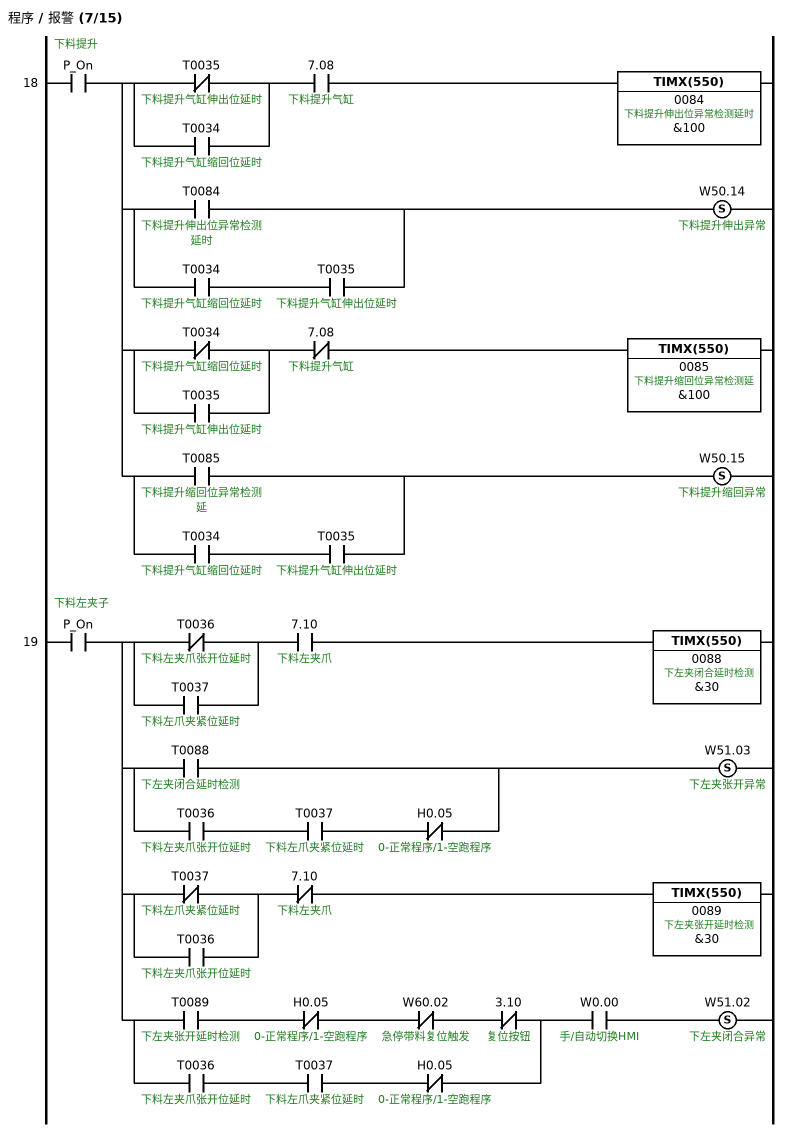
; rung 18: 下料提升
LD P_On
OUT TR0
LDNOT T0035  ; 下料提升气缸伸出位延时
OR T0034  ; 下料提升气缸缩回位延时
ANDLD
AND 7.08  ; 下料提升气缸
TIMX(550) 0084 &100  ; 下料提升伸出位异常检测延时
LD TR0
LD T0084  ; 下料提升伸出位异常检测延时
LD T0034  ; 下料提升气缸缩回位延时
AND T0035  ; 下料提升气缸伸出位延时
ORLD
ANDLD
SET W50.14  ; 下料提升伸出异常
LD TR0
LDNOT T0034  ; 下料提升气缸缩回位延时
OR T0035  ; 下料提升气缸伸出位延时
ANDLD
ANDNOT 7.08  ; 下料提升气缸
TIMX(550) 0085 &100  ; 下料提升缩回位异常检测延
LD TR0
LD T0085  ; 下料提升缩回位异常检测延
LD T0034  ; 下料提升气缸缩回位延时
AND T0035  ; 下料提升气缸伸出位延时
ORLD
ANDLD
SET W50.15  ; 下料提升缩回异常
; rung 19: 下料左夹子
LD P_On
OUT TR0
LDNOT T0036  ; 下料左夹爪张开位延时
OR T0037  ; 下料左爪夹紧位延时
ANDLD
AND 7.10  ; 下料左夹爪
TIMX(550) 0088 &30  ; 下左夹闭合延时检测
LD TR0
LD T0088  ; 下左夹闭合延时检测
LD T0036  ; 下料左夹爪张开位延时
AND T0037  ; 下料左爪夹紧位延时
ANDNOT H0.05  ; 0-正常程序/1-空跑程序
ORLD
ANDLD
SET W51.03  ; 下左夹张开异常
LD TR0
LDNOT T0037  ; 下料左爪夹紧位延时
OR T0036  ; 下料左夹爪张开位延时
ANDLD
ANDNOT 7.10  ; 下料左夹爪
TIMX(550) 0089 &30  ; 下左夹张开延时检测
LD TR0
LD T0089  ; 下左夹张开延时检测
ANDNOT H0.05  ; 0-正常程序/1-空跑程序
ANDNOT W60.02  ; 急停带料复位触发
ANDNOT 3.10  ; 复位按钮
LD T0036  ; 下料左夹爪张开位延时
AND T0037  ; 下料左爪夹紧位延时
ANDNOT H0.05  ; 0-正常程序/1-空跑程序
ORLD
ANDLD
AND W0.00  ; 手/自动切换HMI
SET W51.02  ; 下左夹闭合异常

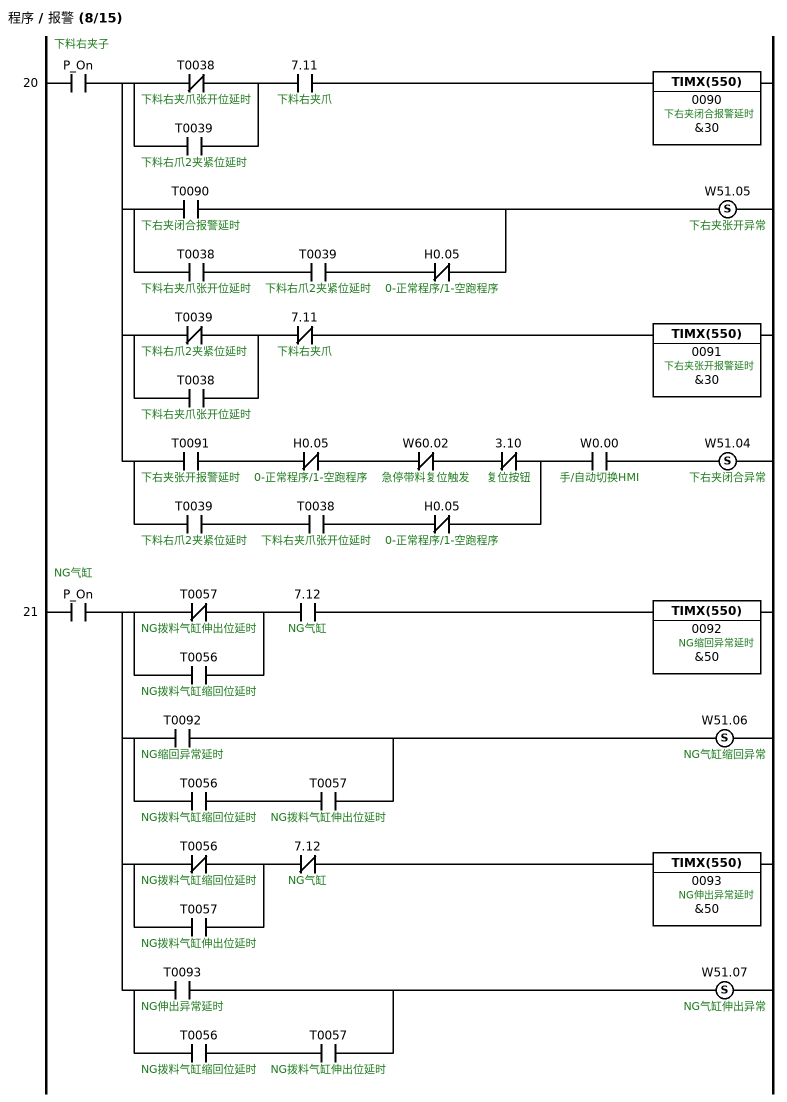
; rung 20: 下料右夹子
LD P_On
OUT TR0
LDNOT T0038  ; 下料右夹爪张开位延时
OR T0039  ; 下料右爪2夹紧位延时
ANDLD
AND 7.11  ; 下料右夹爪
TIMX(550) 0090 &30  ; 下右夹闭合报警延时
LD TR0
LD T0090  ; 下右夹闭合报警延时
LD T0038  ; 下料右夹爪张开位延时
AND T0039  ; 下料右爪2夹紧位延时
ANDNOT H0.05  ; 0-正常程序/1-空跑程序
ORLD
ANDLD
SET W51.05  ; 下右夹张开异常
LD TR0
LDNOT T0039  ; 下料右爪2夹紧位延时
OR T0038  ; 下料右夹爪张开位延时
ANDLD
ANDNOT 7.11  ; 下料右夹爪
TIMX(550) 0091 &30  ; 下右夹张开报警延时
LD TR0
LD T0091  ; 下右夹张开报警延时
ANDNOT H0.05  ; 0-正常程序/1-空跑程序
ANDNOT W60.02  ; 急停带料复位触发
ANDNOT 3.10  ; 复位按钮
LD T0039  ; 下料右爪2夹紧位延时
AND T0038  ; 下料右夹爪张开位延时
ANDNOT H0.05  ; 0-正常程序/1-空跑程序
ORLD
ANDLD
AND W0.00  ; 手/自动切换HMI
SET W51.04  ; 下右夹闭合异常
; rung 21: NG气缸
LD P_On
OUT TR0
LDNOT T0057  ; NG拨料气缸伸出位延时
OR T0056  ; NG拨料气缸缩回位延时
ANDLD
AND 7.12  ; NG气缸
TIMX(550) 0092 &50  ; NG缩回异常延时
LD TR0
LD T0092  ; NG缩回异常延时
LD T0056  ; NG拨料气缸缩回位延时
AND T0057  ; NG拨料气缸伸出位延时
ORLD
ANDLD
SET W51.06  ; NG气缸缩回异常
LD TR0
LDNOT T0056  ; NG拨料气缸缩回位延时
OR T0057  ; NG拨料气缸伸出位延时
ANDLD
ANDNOT 7.12  ; NG气缸
TIMX(550) 0093 &50  ; NG伸出异常延时
LD TR0
LD T0093  ; NG伸出异常延时
LD T0056  ; NG拨料气缸缩回位延时
AND T0057  ; NG拨料气缸伸出位延时
ORLD
ANDLD
SET W51.07  ; NG气缸伸出异常

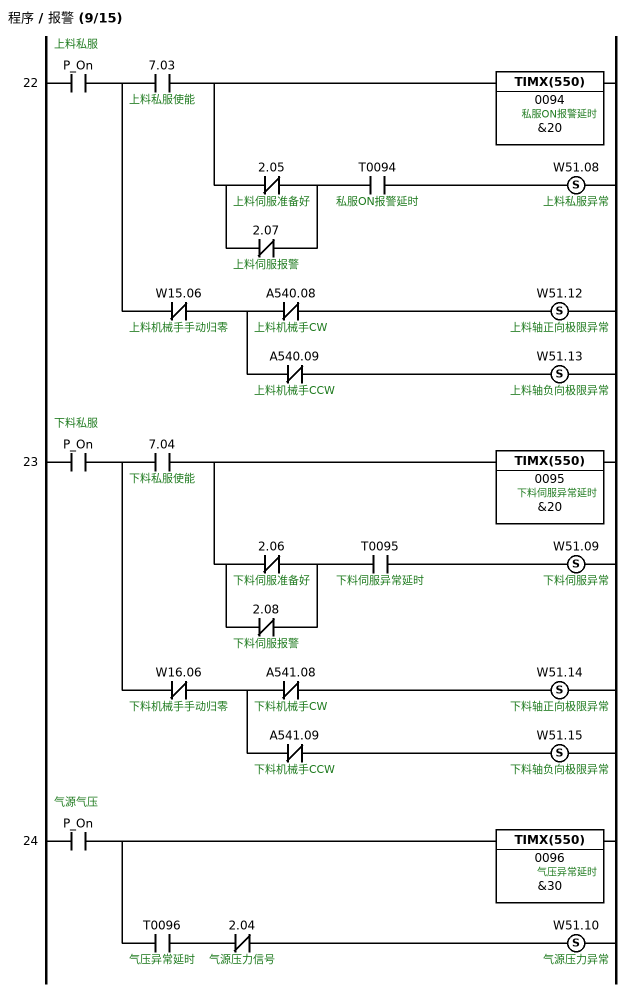
; rung 22: 上料私服
LD P_On
OUT TR0
AND 7.03  ; 上料私服使能
TIMX(550) 0094 &20  ; 私服ON报警延时
LDNOT 2.05  ; 上料伺服准备好
ORNOT 2.07  ; 上料伺服报警
ANDLD
AND T0094  ; 私服ON报警延时
SET W51.08  ; 上料私服异常
LD TR0
ANDNOT W15.06  ; 上料机械手手动归零
OUT TR0
ANDNOT A540.08  ; 上料机械手CW
SET W51.12  ; 上料轴正向极限异常
LD TR0
ANDNOT A540.09  ; 上料机械手CCW
SET W51.13  ; 上料轴负向极限异常
; rung 23: 下料私服
LD P_On
OUT TR0
AND 7.04  ; 下料私服使能
TIMX(550) 0095 &20  ; 下料伺服异常延时
LDNOT 2.06  ; 下料伺服准备好
ORNOT 2.08  ; 下料伺服报警
ANDLD
AND T0095  ; 下料伺服异常延时
SET W51.09  ; 下料伺服异常
LD TR0
ANDNOT W16.06  ; 下料机械手手动归零
OUT TR0
ANDNOT A541.08  ; 下料机械手CW
SET W51.14  ; 下料轴正向极限异常
LD TR0
ANDNOT A541.09  ; 下料机械手CCW
SET W51.15  ; 下料轴负向极限异常
; rung 24: 气源气压
LD P_On
TIMX(550) 0096 &30  ; 气压异常延时
AND T0096  ; 气压异常延时
ANDNOT 2.04  ; 气源压力信号
SET W51.10  ; 气源压力异常

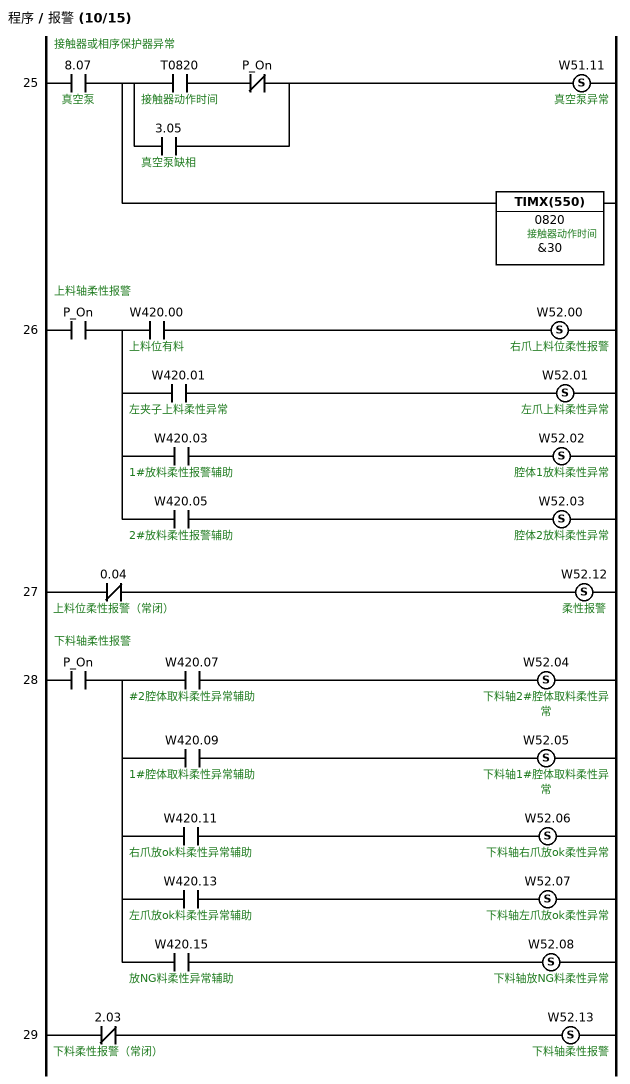
; rung 25: 接触器或相序保护器异常
LD 8.07  ; 真空泵
OUT TR0
LD T0820  ; 接触器动作时间
ANDNOT P_On
OR 3.05  ; 真空泵缺相
ANDLD
SET W51.11  ; 真空泵异常
LD TR0
TIMX(550) 0820 &30  ; 接触器动作时间
; rung 26: 上料轴柔性报警
LD P_On
OUT TR0
AND W420.00  ; 上料位有料
SET W52.00  ; 右爪上料位柔性报警
LD TR0
AND W420.01  ; 左夹子上料柔性异常
SET W52.01  ; 左爪上料柔性异常
LD TR0
AND W420.03  ; 1#放料柔性报警辅助
SET W52.02  ; 腔体1放料柔性异常
LD TR0
AND W420.05  ; 2#放料柔性报警辅助
SET W52.03  ; 腔体2放料柔性异常
; rung 27
LDNOT 0.04  ; 上料位柔性报警（常闭）
SET W52.12  ; 柔性报警
; rung 28: 下料轴柔性报警
LD P_On
OUT TR0
AND W420.07  ; #2腔体取料柔性异常辅助
SET W52.04  ; 下料轴2#腔体取料柔性异常
LD TR0
AND W420.09  ; 1#腔体取料柔性异常辅助
SET W52.05  ; 下料轴1#腔体取料柔性异常
LD TR0
AND W420.11  ; 右爪放ok料柔性异常辅助
SET W52.06  ; 下料轴右爪放ok柔性异常
LD TR0
AND W420.13  ; 左爪放ok料柔性异常辅助
SET W52.07  ; 下料轴左爪放ok柔性异常
LD TR0
AND W420.15  ; 放NG料柔性异常辅助
SET W52.08  ; 下料轴放NG料柔性异常
; rung 29
LDNOT 2.03  ; 下料柔性报警（常闭）
SET W52.13  ; 下料轴柔性报警

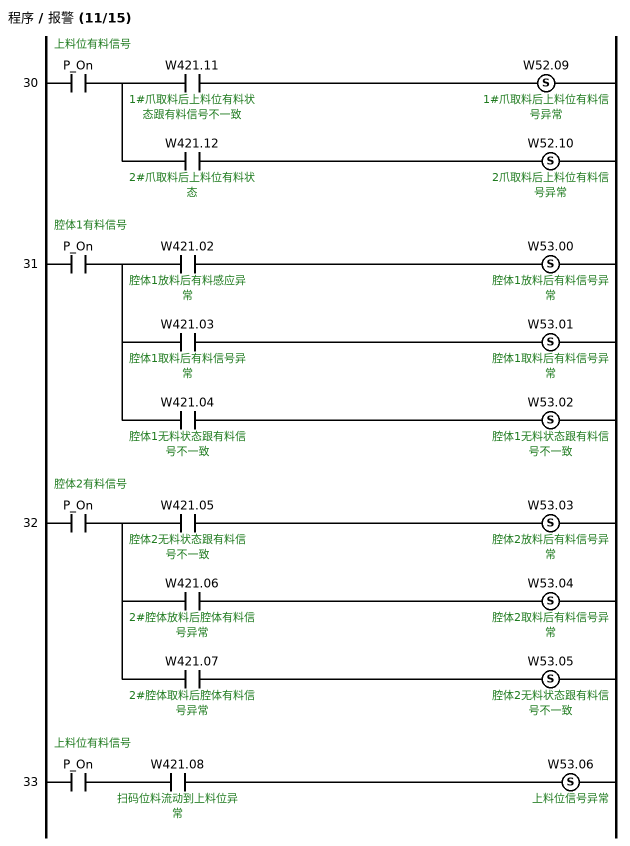
; rung 30: 上料位有料信号
LD P_On
OUT TR0
AND W421.11  ; 1#爪取料后上料位有料状态跟有料信号不一致
SET W52.09  ; 1#爪取料后上料位有料信号异常
LD TR0
AND W421.12  ; 2#爪取料后上料位有料状态
SET W52.10  ; 2爪取料后上料位有料信号异常
; rung 31: 腔体1有料信号
LD P_On
OUT TR0
AND W421.02  ; 腔体1放料后有料感应异常
SET W53.00  ; 腔体1放料后有料信号异常
LD TR0
AND W421.03  ; 腔体1取料后有料信号异常
SET W53.01  ; 腔体1取料后有料信号异常
LD TR0
AND W421.04  ; 腔体1无料状态跟有料信号不一致
SET W53.02  ; 腔体1无料状态跟有料信号不一致
; rung 32: 腔体2有料信号
LD P_On
OUT TR0
AND W421.05  ; 腔体2无料状态跟有料信号不一致
SET W53.03  ; 腔体2放料后有料信号异常
LD TR0
AND W421.06  ; 2#腔体放料后腔体有料信号异常
SET W53.04  ; 腔体2取料后有料信号异常
LD TR0
AND W421.07  ; 2#腔体取料后腔体有料信号异常
SET W53.05  ; 腔体2无料状态跟有料信号不一致
; rung 33: 上料位有料信号
LD P_On
AND W421.08  ; 扫码位料流动到上料位异常
SET W53.06  ; 上料位信号异常

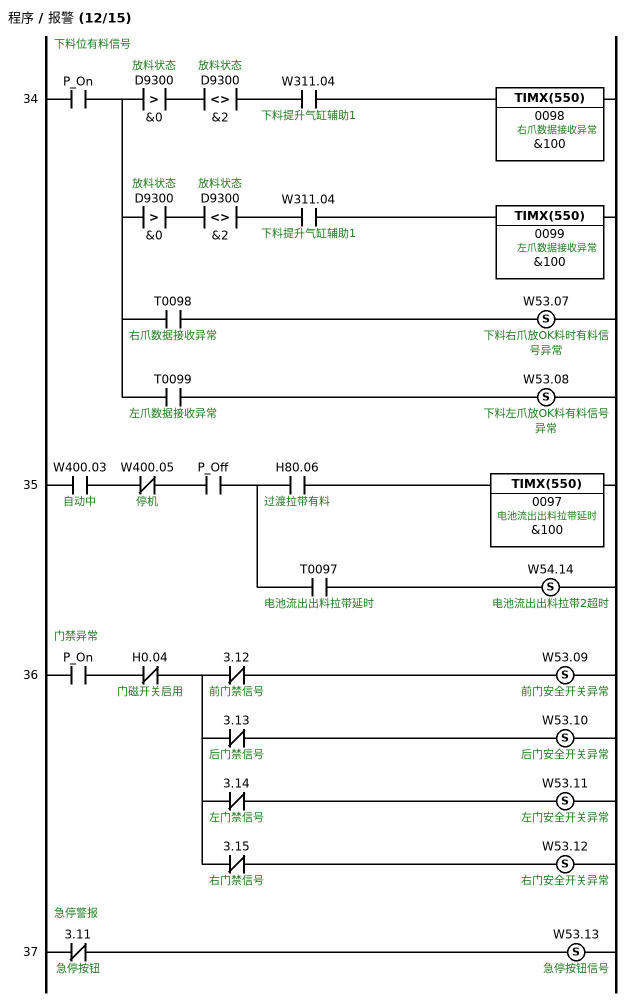
; rung 34: 下料位有料信号
LD P_On
OUT TR0
AND>(320) D9300 &0  ; 放料状态
AND<>(305) D9300 &2  ; 放料状态
AND W311.04  ; 下料提升气缸辅助1
TIMX(550) 0098 &100  ; 右爪数据接收异常
LD TR0
AND>(320) D9300 &0  ; 放料状态
AND<>(305) D9300 &2  ; 放料状态
AND W311.04  ; 下料提升气缸辅助1
TIMX(550) 0099 &100  ; 左爪数据接收异常
LD TR0
AND T0098  ; 右爪数据接收异常
SET W53.07  ; 下料右爪放OK料时有料信号异常
LD TR0
AND T0099  ; 左爪数据接收异常
SET W53.08  ; 下料左爪放OK料有料信号异常
; rung 35
LD W400.03  ; 自动中
ANDNOT W400.05  ; 停机
AND P_Off
OUT TR0
AND H80.06  ; 过渡拉带有料
TIMX(550) 0097 &100  ; 电池流出出料拉带延时
LD TR0
AND T0097  ; 电池流出出料拉带延时
SET W54.14  ; 电池流出出料拉带2超时
; rung 36: 门禁异常
LD P_On
ANDNOT H0.04  ; 门磁开关启用
OUT TR0
ANDNOT 3.12  ; 前门禁信号
SET W53.09  ; 前门安全开关异常
LD TR0
ANDNOT 3.13  ; 后门禁信号
SET W53.10  ; 后门安全开关异常
LD TR0
ANDNOT 3.14  ; 左门禁信号
SET W53.11  ; 左门安全开关异常
LD TR0
ANDNOT 3.15  ; 右门禁信号
SET W53.12  ; 右门安全开关异常
; rung 37: 急停警报
LDNOT 3.11  ; 急停按钮
SET W53.13  ; 急停按钮信号

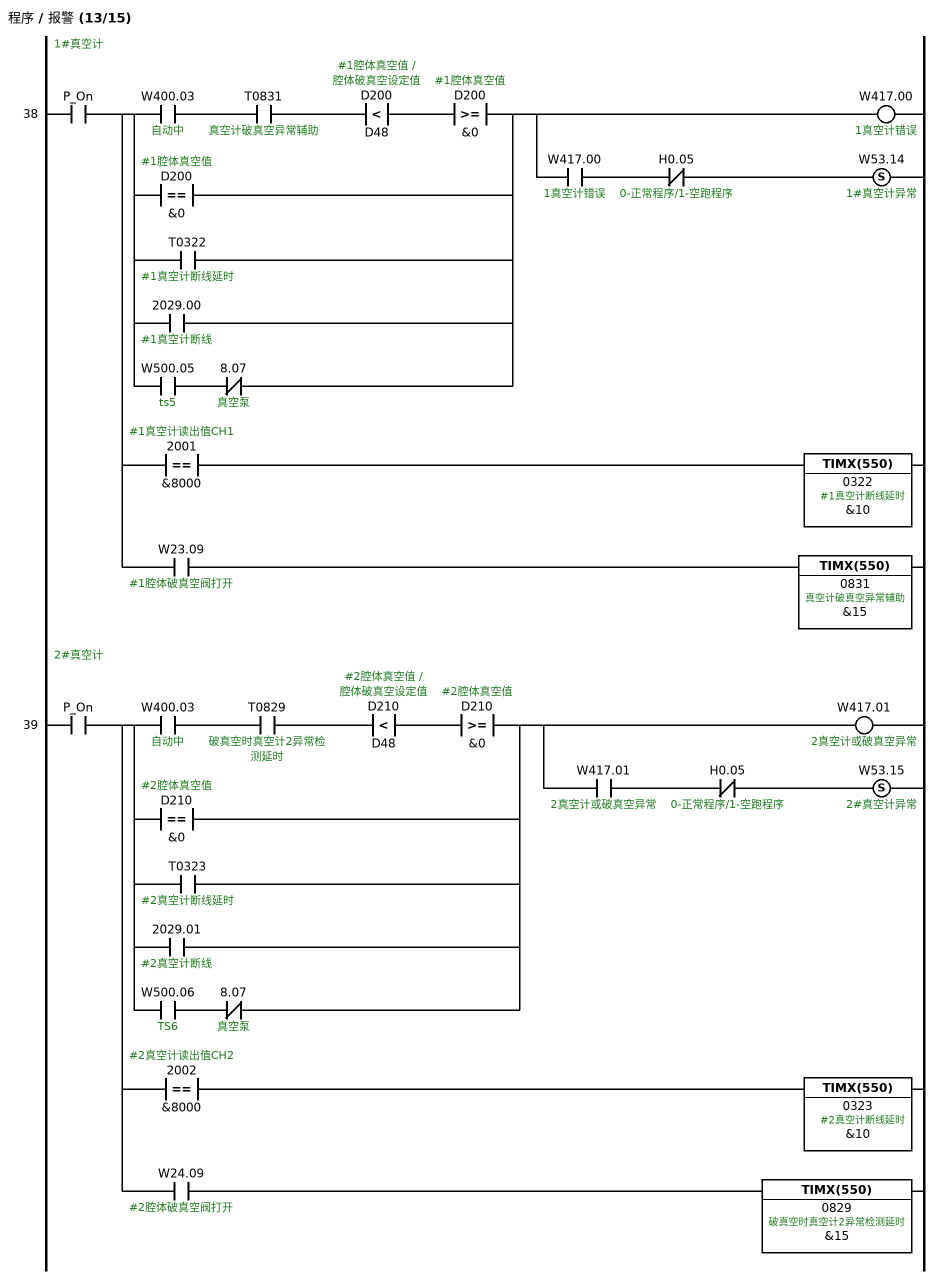
; rung 38: 1#真空计
LD P_On
OUT TR0
LD W400.03  ; 自动中
AND T0831  ; 真空计破真空异常辅助
AND<F(331) D200 D48  ; #1腔体真空值, 腔体破真空设定值
AND>=F(334) D200 &0  ; #1腔体真空值
OR=F(329) D200 &0  ; #1腔体真空值
OR T0322  ; #1真空计断线延时
OR 2029.00  ; #1真空计断线
LD W500.05  ; ts5
ANDNOT 8.07  ; 真空泵
ORLD
ANDLD
OUT W417.00  ; 1真空计错误
AND W417.00  ; 1真空计错误
ANDNOT H0.05  ; 0-正常程序/1-空跑程序
SET W53.14  ; 1#真空计异常
LD TR0
AND=(300) 2001 &8000  ; #1真空计读出值CH1
TIMX(550) 0322 &10  ; #1真空计断线延时
LD TR0
AND W23.09  ; #1腔体破真空阀打开
TIMX(550) 0831 &15  ; 真空计破真空异常辅助
; rung 39: 2#真空计
LD P_On
OUT TR0
LD W400.03  ; 自动中
AND T0829  ; 破真空时真空计2异常检测延时
AND<F(331) D210 D48  ; #2腔体真空值, 腔体破真空设定值
AND>=F(334) D210 &0  ; #2腔体真空值
OR=F(329) D210 &0  ; #2腔体真空值
OR T0323  ; #2真空计断线延时
OR 2029.01  ; #2真空计断线
LD W500.06  ; TS6
ANDNOT 8.07  ; 真空泵
ORLD
ANDLD
OUT W417.01  ; 2真空计或破真空异常
AND W417.01  ; 2真空计或破真空异常
ANDNOT H0.05  ; 0-正常程序/1-空跑程序
SET W53.15  ; 2#真空计异常
LD TR0
AND=(300) 2002 &8000  ; #2真空计读出值CH2
TIMX(550) 0323 &10  ; #2真空计断线延时
LD TR0
AND W24.09  ; #2腔体破真空阀打开
TIMX(550) 0829 &15  ; 破真空时真空计2异常检测延时

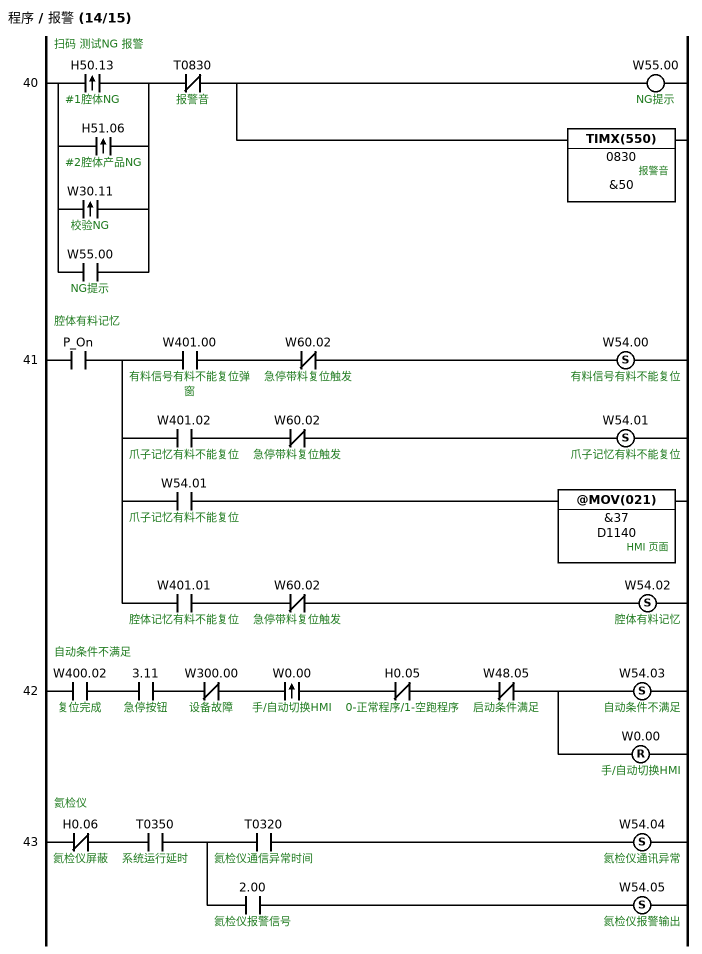
; rung 40: 扫码 测试NG 报警
@LD H50.13  ; #1腔体NG
@OR H51.06  ; #2腔体产品NG
@OR W30.11  ; 校验NG
OR W55.00  ; NG提示
ANDNOT T0830  ; 报警音
OUT W55.00  ; NG提示
TIMX(550) 0830 &50  ; 报警音
; rung 41: 腔体有料记忆
LD P_On
OUT TR0
AND W401.00  ; 有料信号有料不能复位弹窗
ANDNOT W60.02  ; 急停带料复位触发
SET W54.00  ; 有料信号有料不能复位
LD TR0
AND W401.02  ; 爪子记忆有料不能复位
ANDNOT W60.02  ; 急停带料复位触发
SET W54.01  ; 爪子记忆有料不能复位
LD TR0
AND W54.01  ; 爪子记忆有料不能复位
@MOV(021) &37 D1140  ; HMI 页面
LD TR0
AND W401.01  ; 腔体记忆有料不能复位
ANDNOT W60.02  ; 急停带料复位触发
SET W54.02  ; 腔体有料记忆
; rung 42: 自动条件不满足
LD W400.02  ; 复位完成
AND 3.11  ; 急停按钮
ANDNOT W300.00  ; 设备故障
@AND W0.00  ; 手/自动切换HMI
ANDNOT H0.05  ; 0-正常程序/1-空跑程序
ANDNOT W48.05  ; 启动条件满足
SET W54.03  ; 自动条件不满足
RSET W0.00  ; 手/自动切换HMI
; rung 43: 氦检仪
LDNOT H0.06  ; 氦检仪屏蔽
AND T0350  ; 系统运行延时  // 2018/7/25 由常通改为T350，避免开机氦检仪报警
OUT TR0
AND T0320  ; 氦检仪通信异常时间
SET W54.04  ; 氦检仪通讯异常
LD TR0
AND 2.00  ; 氦检仪报警信号
SET W54.05  ; 氦检仪报警输出

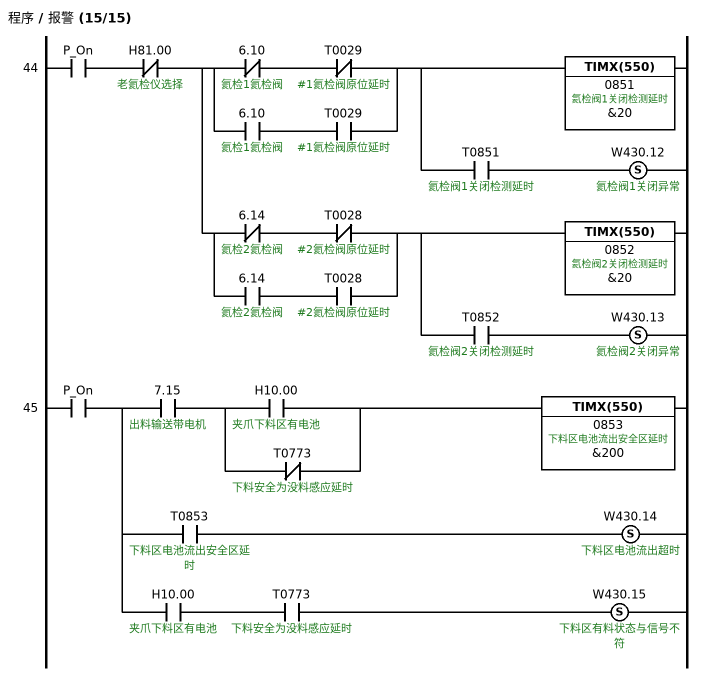
; rung 44
LD P_On
ANDNOT H81.00  ; 老氦检仪选择
OUT TR0
LDNOT 6.10  ; 氦检1氦检阀
ANDNOT T0029  ; #1氦检阀原位延时
LD 6.10  ; 氦检1氦检阀
AND T0029  ; #1氦检阀原位延时
ORLD
ANDLD
TIMX(550) 0851 &20  ; 氦检阀1关闭检测延时
AND T0851  ; 氦检阀1关闭检测延时
SET W430.12  ; 氦检阀1关闭异常
LD TR0
LDNOT 6.14  ; 氦检2氦检阀
ANDNOT T0028  ; #2氦检阀原位延时
LD 6.14  ; 氦检2氦检阀
AND T0028  ; #2氦检阀原位延时
ORLD
ANDLD
TIMX(550) 0852 &20  ; 氦检阀2关闭检测延时
AND T0852  ; 氦检阀2关闭检测延时
SET W430.13  ; 氦检阀2关闭异常
; rung 45
LD P_On
OUT TR0
AND 7.15  ; 出料输送带电机
LD H10.00  ; 夹爪下料区有电池
ORNOT T0773  ; 下料安全为没料感应延时
ANDLD
TIMX(550) 0853 &200  ; 下料区电池流出安全区延时
LD TR0
AND T0853  ; 下料区电池流出安全区延时
SET W430.14  ; 下料区电池流出超时
LD TR0
AND H10.00  ; 夹爪下料区有电池
AND T0773  ; 下料安全为没料感应延时
SET W430.15  ; 下料区有料状态与信号不符

### Section 传感器屏蔽及延时

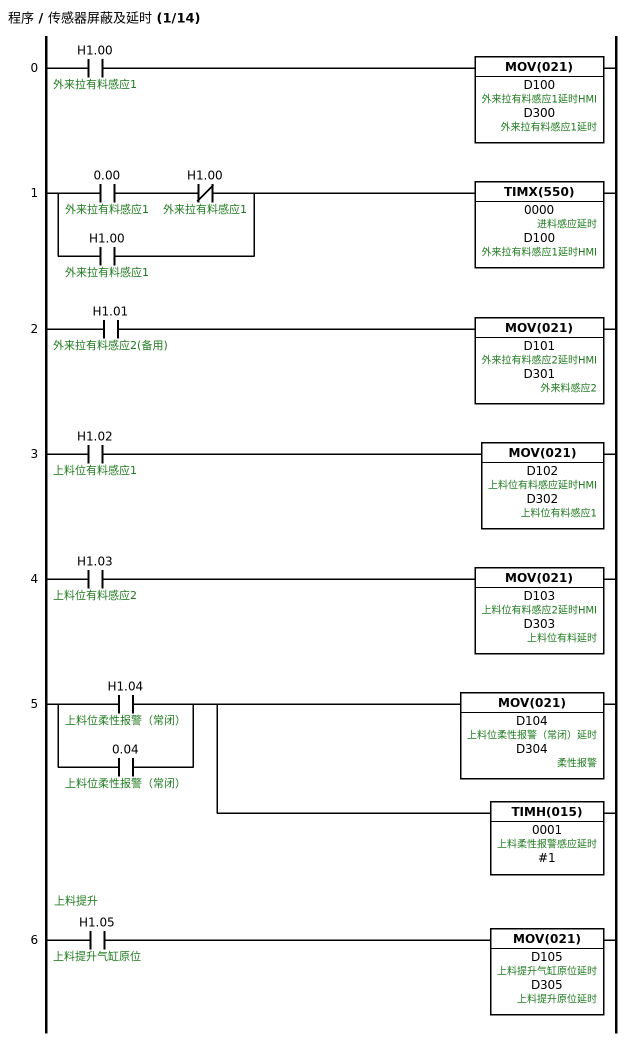
; rung 0
LD H1.00  ; 外来拉有料感应1
MOV(021) D100 D300  ; 外来拉有料感应1延时HMI, 外来拉有料感应1延时
; rung 1
LD 0.00  ; 外来拉有料感应1
ANDNOT H1.00  ; 外来拉有料感应1
OR H1.00  ; 外来拉有料感应1
TIMX(550) 0000 D100  ; 外来拉有料感应1延时HMI, 进料感应延时
; rung 2
LD H1.01  ; 外来拉有料感应2(备用)
MOV(021) D101 D301  ; 外来拉有料感应2延时HMI, 外来料感应2
; rung 3
LD H1.02  ; 上料位有料感应1
MOV(021) D102 D302  ; 上料位有料感应延时HMI, 上料位有料感应1
; rung 4
LD H1.03  ; 上料位有料感应2
MOV(021) D103 D303  ; 上料位有料感应2延时HMI, 上料位有料延时
; rung 5
LD H1.04  ; 上料位柔性报警（常闭）
OR 0.04  ; 上料位柔性报警（常闭）
MOV(021) D104 D304  ; 上料位柔性报警（常闭）延时, 柔性报警
TIMH(015) 0001 #1  ; 上料柔性报警感应延时
; rung 6: 上料提升
LD H1.05  ; 上料提升气缸原位
MOV(021) D105 D305  ; 上料提升气缸原位延时, 上料提升原位延时

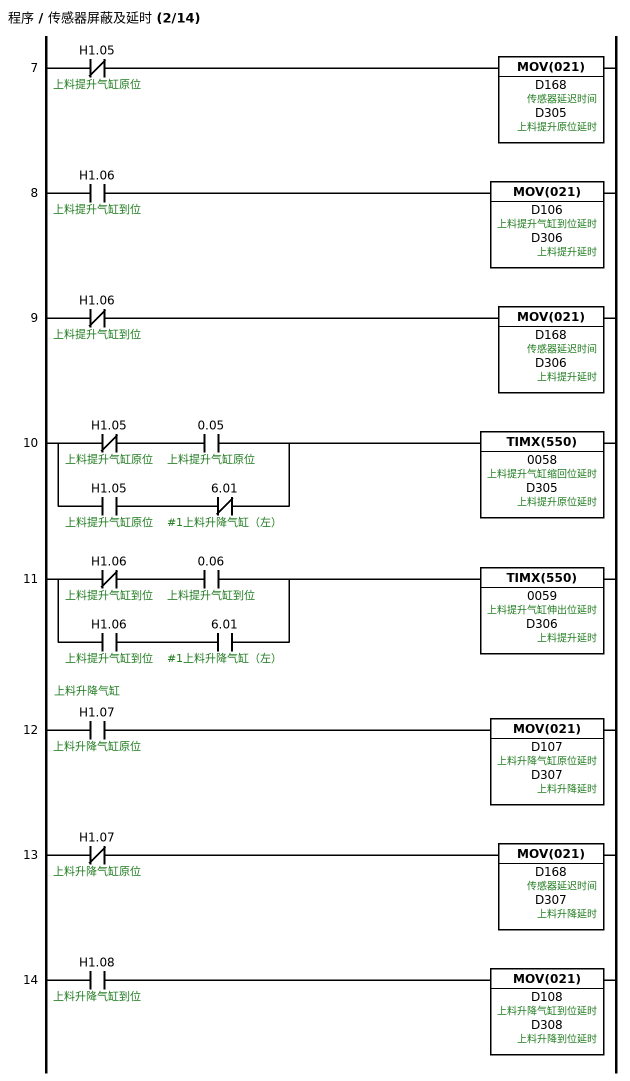
; rung 7
LDNOT H1.05  ; 上料提升气缸原位
MOV(021) D168 D305  ; 传感器延迟时间, 上料提升原位延时
; rung 8
LD H1.06  ; 上料提升气缸到位
MOV(021) D106 D306  ; 上料提升气缸到位延时, 上料提升延时
; rung 9
LDNOT H1.06  ; 上料提升气缸到位
MOV(021) D168 D306  ; 传感器延迟时间, 上料提升延时
; rung 10
LDNOT H1.05  ; 上料提升气缸原位
AND 0.05  ; 上料提升气缸原位
LD H1.05  ; 上料提升气缸原位
ANDNOT 6.01  ; #1上料升降气缸（左）
ORLD
TIMX(550) 0058 D305  ; 上料提升原位延时, 上料提升气缸缩回位延时
; rung 11
LDNOT H1.06  ; 上料提升气缸到位
AND 0.06  ; 上料提升气缸到位
LD H1.06  ; 上料提升气缸到位
AND 6.01  ; #1上料升降气缸（左）
ORLD
TIMX(550) 0059 D306  ; 上料提升延时, 上料提升气缸伸出位延时
; rung 12: 上料升降气缸
LD H1.07  ; 上料升降气缸原位
MOV(021) D107 D307  ; 上料升降气缸原位延时, 上料升降延时
; rung 13
LDNOT H1.07  ; 上料升降气缸原位
MOV(021) D168 D307  ; 传感器延迟时间, 上料升降延时
; rung 14
LD H1.08  ; 上料升降气缸到位
MOV(021) D108 D308  ; 上料升降气缸到位延时, 上料升降到位延时

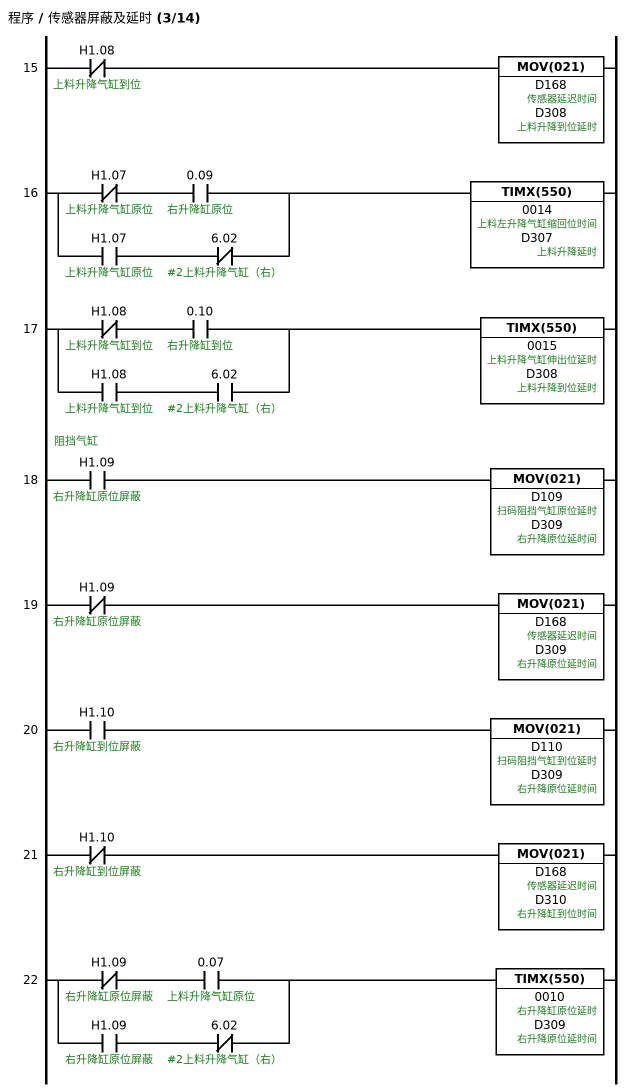
; rung 15
LDNOT H1.08  ; 上料升降气缸到位
MOV(021) D168 D308  ; 传感器延迟时间, 上料升降到位延时
; rung 16
LDNOT H1.07  ; 上料升降气缸原位
AND 0.09  ; 右升降缸原位
LD H1.07  ; 上料升降气缸原位
ANDNOT 6.02  ; #2上料升降气缸（右）
ORLD
TIMX(550) 0014 D307  ; 上料升降延时, 上料左升降气缸缩回位时间
; rung 17
LDNOT H1.08  ; 上料升降气缸到位
AND 0.10  ; 右升降缸到位
LD H1.08  ; 上料升降气缸到位
AND 6.02  ; #2上料升降气缸（右）
ORLD
TIMX(550) 0015 D308  ; 上料升降到位延时, 上料升降气缸伸出位延时
; rung 18: 阻挡气缸
LD H1.09  ; 右升降缸原位屏蔽
MOV(021) D109 D309  ; 扫码阻挡气缸原位延时, 右升降原位延时间
; rung 19
LDNOT H1.09  ; 右升降缸原位屏蔽
MOV(021) D168 D309  ; 传感器延迟时间, 右升降原位延时间
; rung 20
LD H1.10  ; 右升降缸到位屏蔽
MOV(021) D110 D309  ; 扫码阻挡气缸到位延时, 右升降原位延时间
; rung 21
LDNOT H1.10  ; 右升降缸到位屏蔽
MOV(021) D168 D310  ; 传感器延迟时间, 右升降缸到位时间
; rung 22
LDNOT H1.09  ; 右升降缸原位屏蔽
AND 0.07  ; 上料升降气缸原位
LD H1.09  ; 右升降缸原位屏蔽
ANDNOT 6.02  ; #2上料升降气缸（右）
ORLD
TIMX(550) 0010 D309  ; 右升降原位延时间, 右升降缸原位延时

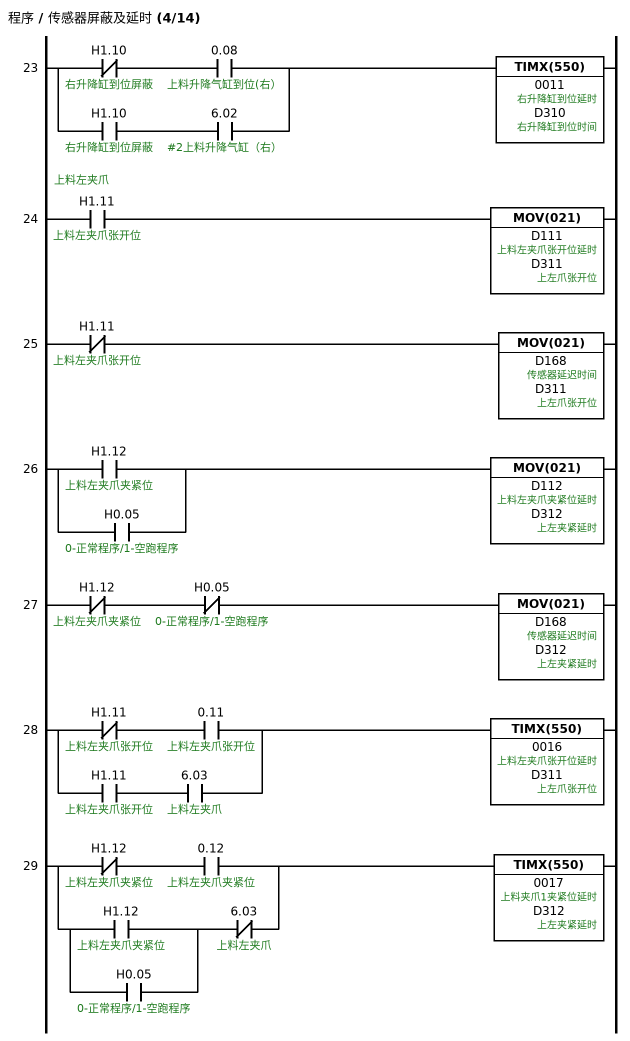
; rung 23
LDNOT H1.10  ; 右升降缸到位屏蔽
AND 0.08  ; 上料升降气缸到位(右）
LD H1.10  ; 右升降缸到位屏蔽
AND 6.02  ; #2上料升降气缸（右）
ORLD
TIMX(550) 0011 D310  ; 右升降缸到位时间, 右升降缸到位延时
; rung 24: 上料左夹爪
LD H1.11  ; 上料左夹爪张开位
MOV(021) D111 D311  ; 上料左夹爪张开位延时, 上左爪张开位
; rung 25
LDNOT H1.11  ; 上料左夹爪张开位
MOV(021) D168 D311  ; 传感器延迟时间, 上左爪张开位
; rung 26
LD H1.12  ; 上料左夹爪夹紧位
OR H0.05  ; 0-正常程序/1-空跑程序
MOV(021) D112 D312  ; 上料左夹爪夹紧位延时, 上左夹紧延时
; rung 27
LDNOT H1.12  ; 上料左夹爪夹紧位
ANDNOT H0.05  ; 0-正常程序/1-空跑程序
MOV(021) D168 D312  ; 传感器延迟时间, 上左夹紧延时
; rung 28
LDNOT H1.11  ; 上料左夹爪张开位
AND 0.11  ; 上料左夹爪张开位
LD H1.11  ; 上料左夹爪张开位
AND 6.03  ; 上料左夹爪
ORLD
TIMX(550) 0016 D311  ; 上左爪张开位, 上料左夹爪张开位延时
; rung 29
LDNOT H1.12  ; 上料左夹爪夹紧位
AND 0.12  ; 上料左夹爪夹紧位
LD H1.12  ; 上料左夹爪夹紧位
OR H0.05  ; 0-正常程序/1-空跑程序
ANDNOT 6.03  ; 上料左夹爪
ORLD
TIMX(550) 0017 D312  ; 上左夹紧延时, 上料夹爪1夹紧位延时

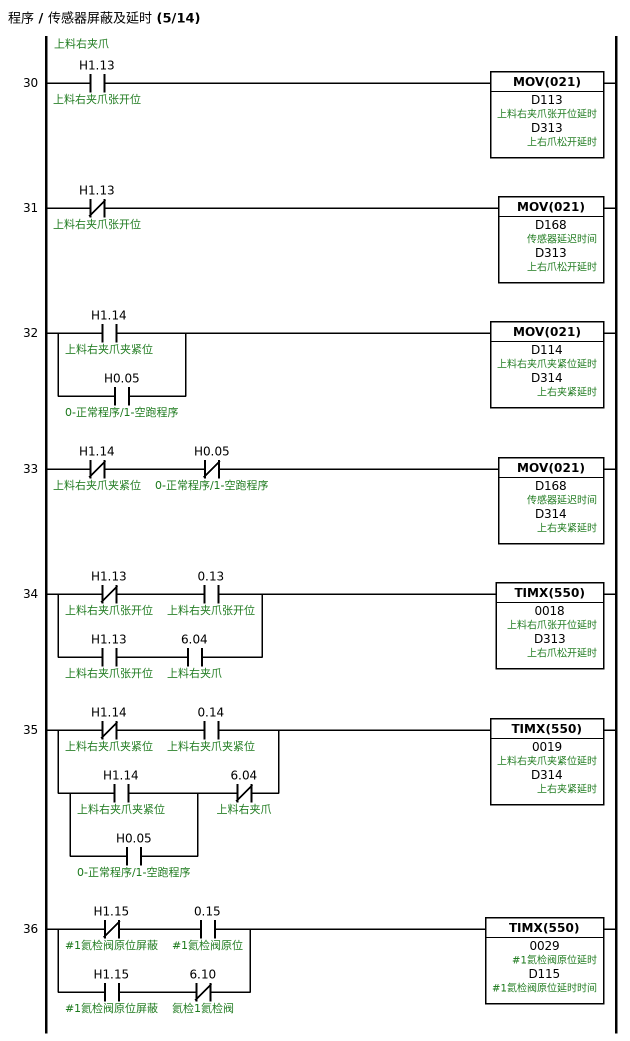
; rung 30: 上料右夹爪
LD H1.13  ; 上料右夹爪张开位
MOV(021) D113 D313  ; 上料右夹爪张开位延时, 上右爪松开延时
; rung 31
LDNOT H1.13  ; 上料右夹爪张开位
MOV(021) D168 D313  ; 传感器延迟时间, 上右爪松开延时
; rung 32
LD H1.14  ; 上料右夹爪夹紧位
OR H0.05  ; 0-正常程序/1-空跑程序
MOV(021) D114 D314  ; 上料右夹爪夹紧位延时, 上右夹紧延时
; rung 33
LDNOT H1.14  ; 上料右夹爪夹紧位
ANDNOT H0.05  ; 0-正常程序/1-空跑程序
MOV(021) D168 D314  ; 传感器延迟时间, 上右夹紧延时
; rung 34
LDNOT H1.13  ; 上料右夹爪张开位
AND 0.13  ; 上料右夹爪张开位
LD H1.13  ; 上料右夹爪张开位
AND 6.04  ; 上料右夹爪
ORLD
TIMX(550) 0018 D313  ; 上右爪松开延时, 上料右爪张开位延时
; rung 35
LDNOT H1.14  ; 上料右夹爪夹紧位
AND 0.14  ; 上料右夹爪夹紧位
LD H1.14  ; 上料右夹爪夹紧位
OR H0.05  ; 0-正常程序/1-空跑程序
ANDNOT 6.04  ; 上料右夹爪
ORLD
TIMX(550) 0019 D314  ; 上右夹紧延时, 上料右夹爪夹紧位延时
; rung 36
LDNOT H1.15  ; #1氦检阀原位屏蔽
AND 0.15  ; #1氦检阀原位
LD H1.15  ; #1氦检阀原位屏蔽
ANDNOT 6.10  ; 氦检1氦检阀
ORLD
TIMX(550) 0029 D115  ; #1氦检阀原位延时时间, #1氦检阀原位延时

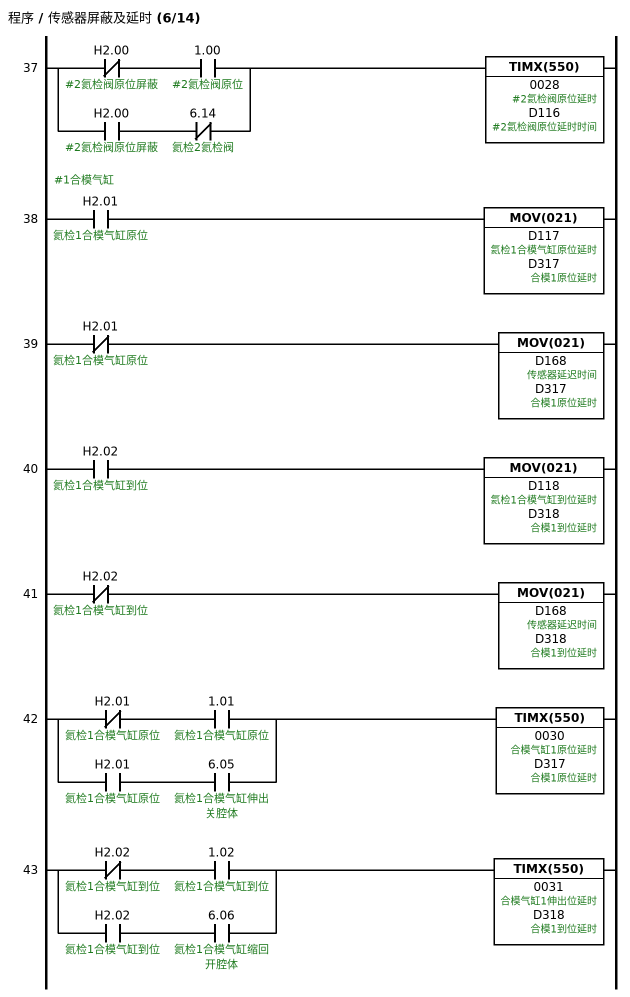
; rung 37
LDNOT H2.00  ; #2氦检阀原位屏蔽
AND 1.00  ; #2氦检阀原位
LD H2.00  ; #2氦检阀原位屏蔽
ANDNOT 6.14  ; 氦检2氦检阀
ORLD
TIMX(550) 0028 D116  ; #2氦检阀原位延时时间, #2氦检阀原位延时
; rung 38: #1合模气缸
LD H2.01  ; 氦检1合模气缸原位
MOV(021) D117 D317  ; 氦检1合模气缸原位延时, 合模1原位延时
; rung 39
LDNOT H2.01  ; 氦检1合模气缸原位
MOV(021) D168 D317  ; 传感器延迟时间, 合模1原位延时
; rung 40
LD H2.02  ; 氦检1合模气缸到位
MOV(021) D118 D318  ; 氦检1合模气缸到位延时, 合模1到位延时
; rung 41
LDNOT H2.02  ; 氦检1合模气缸到位
MOV(021) D168 D318  ; 传感器延迟时间, 合模1到位延时
; rung 42
LDNOT H2.01  ; 氦检1合模气缸原位
AND 1.01  ; 氦检1合模气缸原位
LD H2.01  ; 氦检1合模气缸原位
AND 6.05  ; 氦检1合模气缸伸出 关腔体
ORLD
TIMX(550) 0030 D317  ; 合模1原位延时, 合模气缸1原位延时
; rung 43
LDNOT H2.02  ; 氦检1合模气缸到位
AND 1.02  ; 氦检1合模气缸到位
LD H2.02  ; 氦检1合模气缸到位
AND 6.06  ; 氦检1合模气缸缩回 开腔体
ORLD
TIMX(550) 0031 D318  ; 合模1到位延时, 合模气缸1伸出位延时

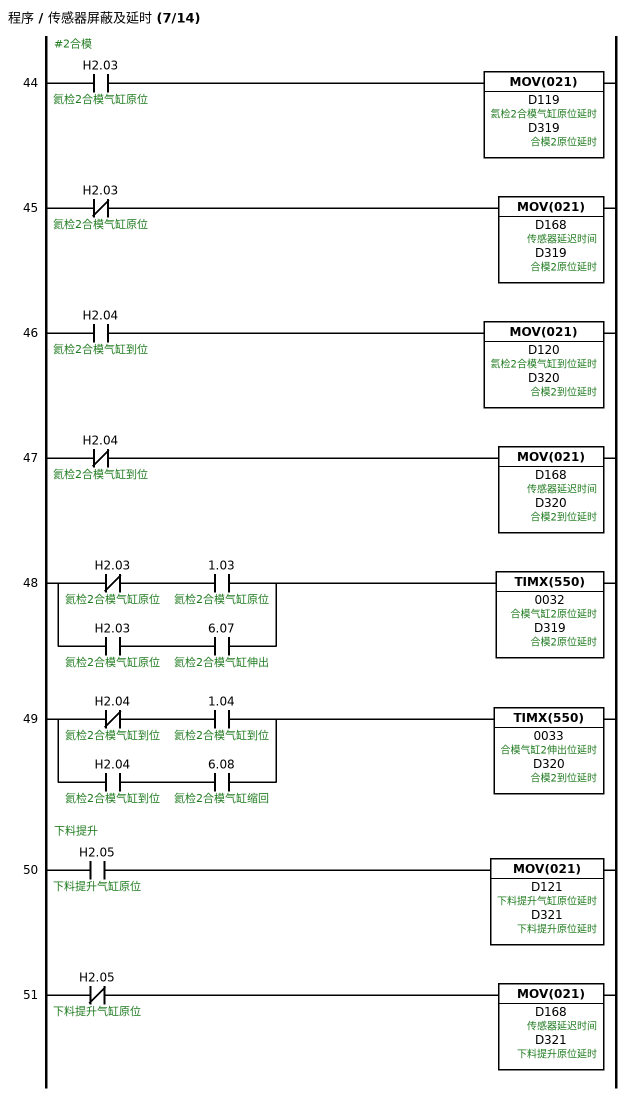
; rung 44: #2合模
LD H2.03  ; 氦检2合模气缸原位
MOV(021) D119 D319  ; 氦检2合模气缸原位延时, 合模2原位延时
; rung 45
LDNOT H2.03  ; 氦检2合模气缸原位
MOV(021) D168 D319  ; 传感器延迟时间, 合模2原位延时
; rung 46
LD H2.04  ; 氦检2合模气缸到位
MOV(021) D120 D320  ; 氦检2合模气缸到位延时, 合模2到位延时
; rung 47
LDNOT H2.04  ; 氦检2合模气缸到位
MOV(021) D168 D320  ; 传感器延迟时间, 合模2到位延时
; rung 48
LDNOT H2.03  ; 氦检2合模气缸原位
AND 1.03  ; 氦检2合模气缸原位
LD H2.03  ; 氦检2合模气缸原位
AND 6.07  ; 氦检2合模气缸伸出
ORLD
TIMX(550) 0032 D319  ; 合模2原位延时, 合模气缸2原位延时
; rung 49
LDNOT H2.04  ; 氦检2合模气缸到位
AND 1.04  ; 氦检2合模气缸到位
LD H2.04  ; 氦检2合模气缸到位
AND 6.08  ; 氦检2合模气缸缩回
ORLD
TIMX(550) 0033 D320  ; 合模2到位延时, 合模气缸2伸出位延时
; rung 50: 下料提升
LD H2.05  ; 下料提升气缸原位
MOV(021) D121 D321  ; 下料提升气缸原位延时, 下料提升原位延时
; rung 51
LDNOT H2.05  ; 下料提升气缸原位
MOV(021) D168 D321  ; 传感器延迟时间, 下料提升原位延时

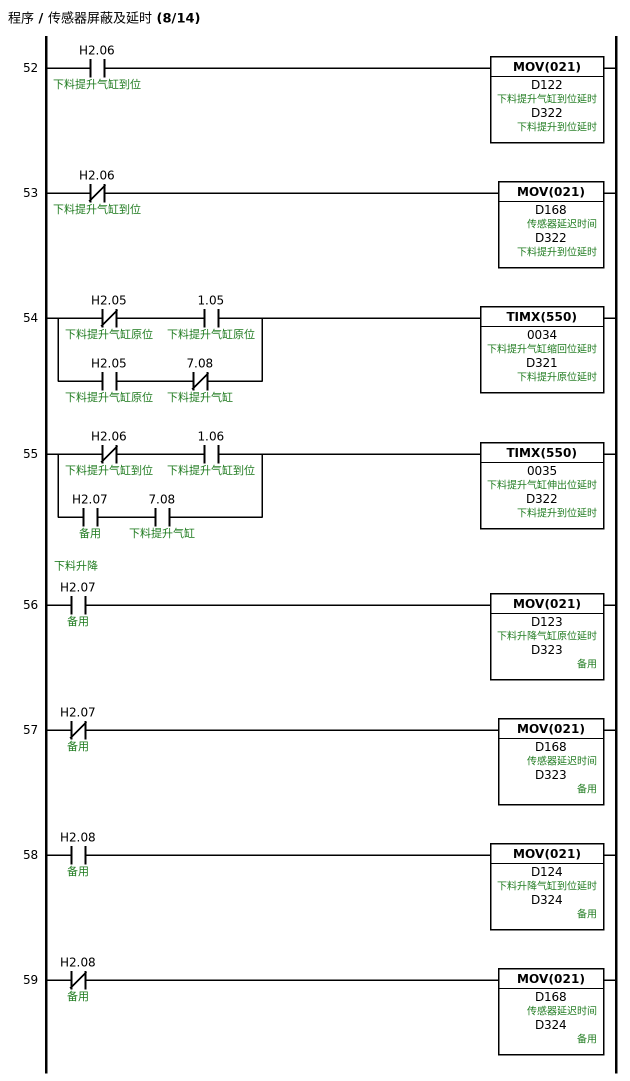
; rung 52
LD H2.06  ; 下料提升气缸到位
MOV(021) D122 D322  ; 下料提升气缸到位延时, 下料提升到位延时
; rung 53
LDNOT H2.06  ; 下料提升气缸到位
MOV(021) D168 D322  ; 传感器延迟时间, 下料提升到位延时
; rung 54
LDNOT H2.05  ; 下料提升气缸原位
AND 1.05  ; 下料提升气缸原位
LD H2.05  ; 下料提升气缸原位
ANDNOT 7.08  ; 下料提升气缸
ORLD
TIMX(550) 0034 D321  ; 下料提升原位延时, 下料提升气缸缩回位延时
; rung 55
LDNOT H2.06  ; 下料提升气缸到位
AND 1.06  ; 下料提升气缸到位
LD H2.07  ; 备用
AND 7.08  ; 下料提升气缸
ORLD
TIMX(550) 0035 D322  ; 下料提升到位延时, 下料提升气缸伸出位延时
; rung 56: 下料升降
LD H2.07  ; 备用
MOV(021) D123 D323  ; 下料升降气缸原位延时, 备用
; rung 57
LDNOT H2.07  ; 备用
MOV(021) D168 D323  ; 传感器延迟时间, 备用
; rung 58
LD H2.08  ; 备用
MOV(021) D124 D324  ; 下料升降气缸到位延时, 备用
; rung 59
LDNOT H2.08  ; 备用
MOV(021) D168 D324  ; 传感器延迟时间, 备用

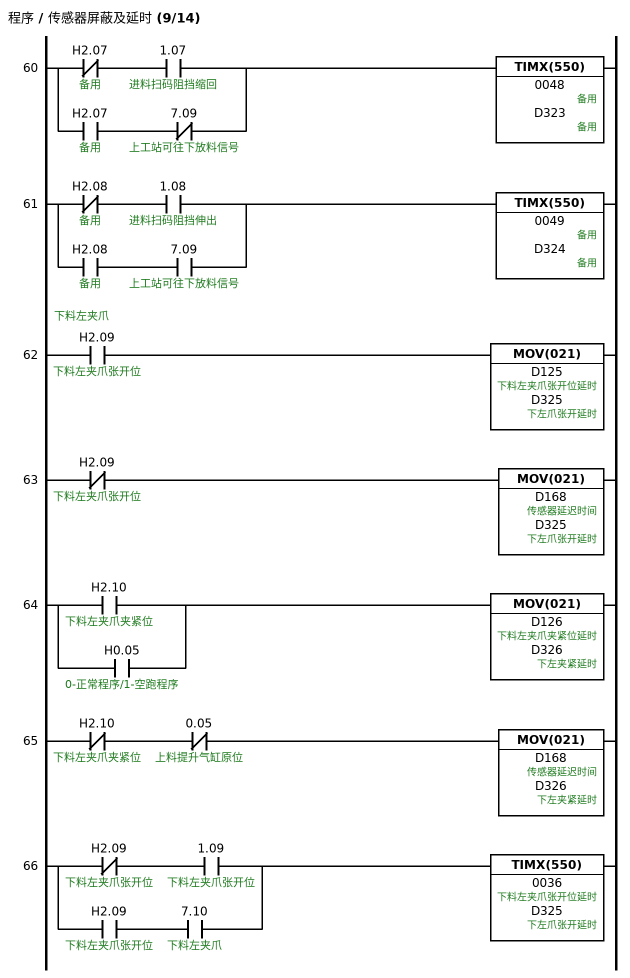
; rung 60
LDNOT H2.07  ; 备用
AND 1.07  ; 进料扫码阻挡缩回
LD H2.07  ; 备用
ANDNOT 7.09  ; 上工站可往下放料信号
ORLD
TIMX(550) 0048 D323  ; 备用
; rung 61
LDNOT H2.08  ; 备用
AND 1.08  ; 进料扫码阻挡伸出
LD H2.08  ; 备用
AND 7.09  ; 上工站可往下放料信号
ORLD
TIMX(550) 0049 D324  ; 备用
; rung 62: 下料左夹爪
LD H2.09  ; 下料左夹爪张开位
MOV(021) D125 D325  ; 下料左夹爪张开位延时, 下左爪张开延时
; rung 63
LDNOT H2.09  ; 下料左夹爪张开位
MOV(021) D168 D325  ; 传感器延迟时间, 下左爪张开延时
; rung 64
LD H2.10  ; 下料左夹爪夹紧位
OR H0.05  ; 0-正常程序/1-空跑程序
MOV(021) D126 D326  ; 下料左夹爪夹紧位延时, 下左夹紧延时
; rung 65
LDNOT H2.10  ; 下料左夹爪夹紧位
ANDNOT 0.05  ; 上料提升气缸原位
MOV(021) D168 D326  ; 传感器延迟时间, 下左夹紧延时
; rung 66
LDNOT H2.09  ; 下料左夹爪张开位
AND 1.09  ; 下料左夹爪张开位
LD H2.09  ; 下料左夹爪张开位
AND 7.10  ; 下料左夹爪
ORLD
TIMX(550) 0036 D325  ; 下左爪张开延时, 下料左夹爪张开位延时

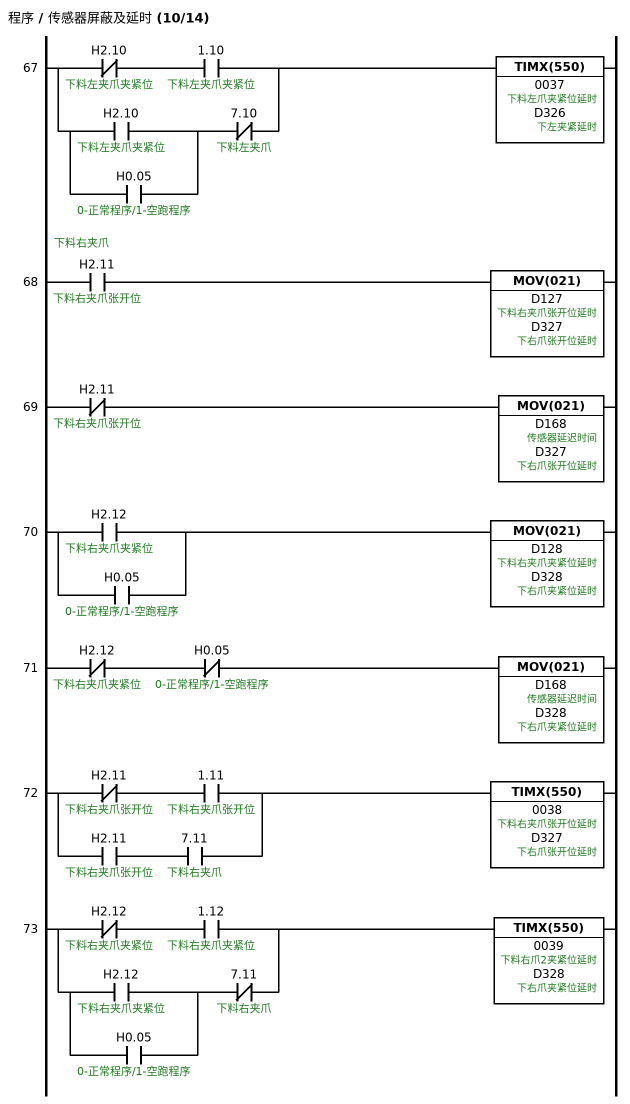
; rung 67
LDNOT H2.10  ; 下料左夹爪夹紧位
AND 1.10  ; 下料左夹爪夹紧位
LD H2.10  ; 下料左夹爪夹紧位
OR H0.05  ; 0-正常程序/1-空跑程序
ANDNOT 7.10  ; 下料左夹爪
ORLD
TIMX(550) 0037 D326  ; 下左夹紧延时, 下料左爪夹紧位延时
; rung 68: 下料右夹爪
LD H2.11  ; 下料右夹爪张开位
MOV(021) D127 D327  ; 下料右夹爪张开位延时, 下右爪张开位延时
; rung 69
LDNOT H2.11  ; 下料右夹爪张开位
MOV(021) D168 D327  ; 传感器延迟时间, 下右爪张开位延时
; rung 70
LD H2.12  ; 下料右夹爪夹紧位
OR H0.05  ; 0-正常程序/1-空跑程序
MOV(021) D128 D328  ; 下料右夹爪夹紧位延时, 下右爪夹紧位延时
; rung 71
LDNOT H2.12  ; 下料右夹爪夹紧位
ANDNOT H0.05  ; 0-正常程序/1-空跑程序
MOV(021) D168 D328  ; 传感器延迟时间, 下右爪夹紧位延时
; rung 72
LDNOT H2.11  ; 下料右夹爪张开位
AND 1.11  ; 下料右夹爪张开位
LD H2.11  ; 下料右夹爪张开位
AND 7.11  ; 下料右夹爪
ORLD
TIMX(550) 0038 D327  ; 下右爪张开位延时, 下料右夹爪张开位延时
; rung 73
LDNOT H2.12  ; 下料右夹爪夹紧位
AND 1.12  ; 下料右夹爪夹紧位
LD H2.12  ; 下料右夹爪夹紧位
OR H0.05  ; 0-正常程序/1-空跑程序
ANDNOT 7.11  ; 下料右夹爪
ORLD
TIMX(550) 0039 D328  ; 下右爪夹紧位延时, 下料右爪2夹紧位延时

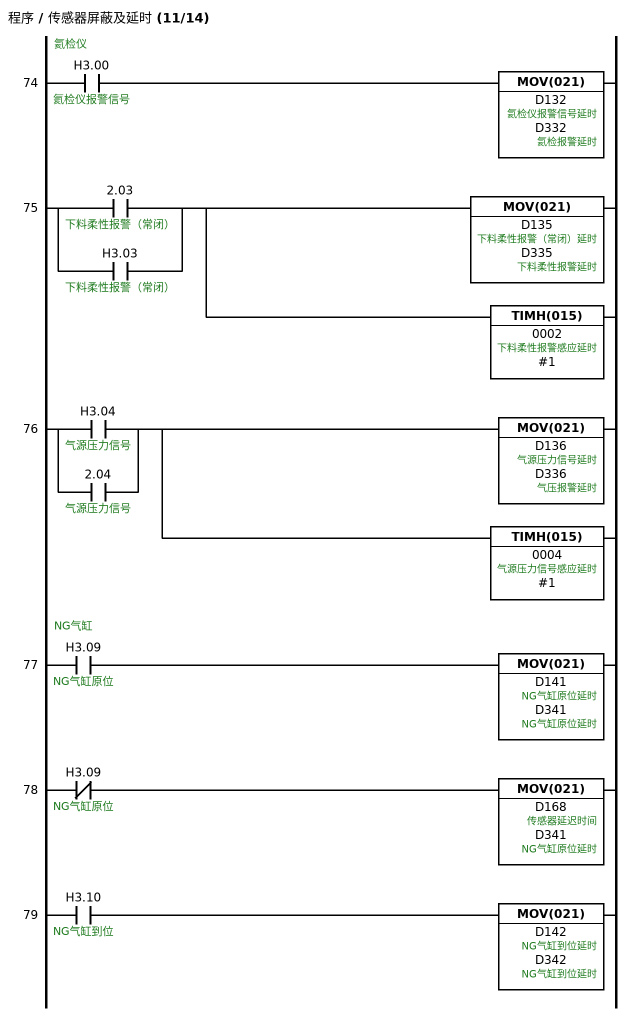
; rung 74: 氦检仪
LD H3.00  ; 氦检仪报警信号
MOV(021) D132 D332  ; 氦检仪报警信号延时, 氦检报警延时
; rung 75
LD 2.03  ; 下料柔性报警（常闭）
OR H3.03  ; 下料柔性报警（常闭）
MOV(021) D135 D335  ; 下料柔性报警（常闭）延时, 下料柔性报警延时
TIMH(015) 0002 #1  ; 下料柔性报警感应延时
; rung 76
LD H3.04  ; 气源压力信号
OR 2.04  ; 气源压力信号
MOV(021) D136 D336  ; 气源压力信号延时, 气压报警延时
TIMH(015) 0004 #1  ; 气源压力信号感应延时
; rung 77: NG气缸
LD H3.09  ; NG气缸原位
MOV(021) D141 D341  ; NG气缸原位延时
; rung 78
LDNOT H3.09  ; NG气缸原位
MOV(021) D168 D341  ; 传感器延迟时间, NG气缸原位延时
; rung 79
LD H3.10  ; NG气缸到位
MOV(021) D142 D342  ; NG气缸到位延时

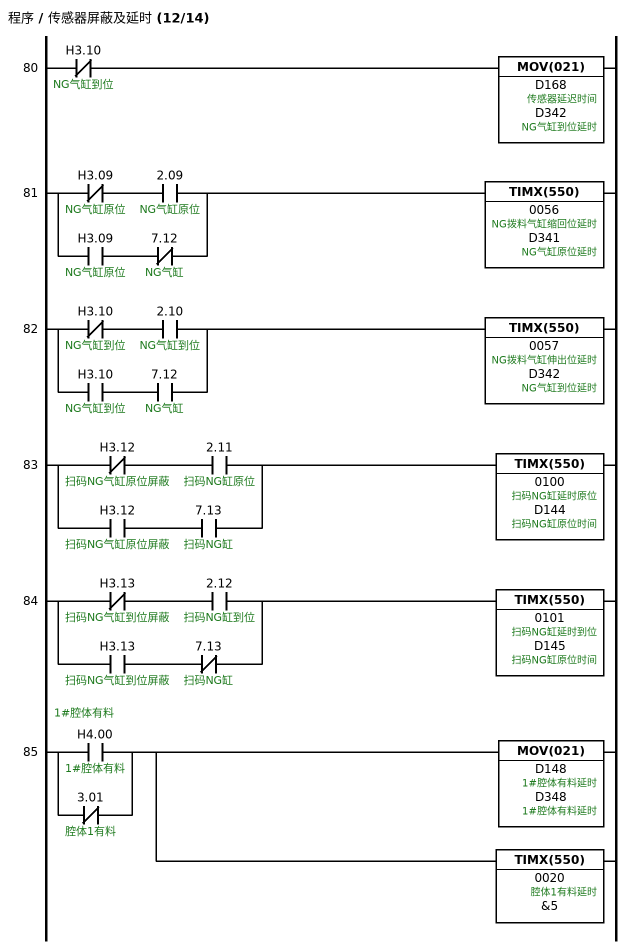
; rung 80
LDNOT H3.10  ; NG气缸到位
MOV(021) D168 D342  ; 传感器延迟时间, NG气缸到位延时
; rung 81
LDNOT H3.09  ; NG气缸原位
AND 2.09  ; NG气缸原位
LD H3.09  ; NG气缸原位
ANDNOT 7.12  ; NG气缸
ORLD
TIMX(550) 0056 D341  ; NG气缸原位延时, NG拨料气缸缩回位延时
; rung 82
LDNOT H3.10  ; NG气缸到位
AND 2.10  ; NG气缸到位
LD H3.10  ; NG气缸到位
AND 7.12  ; NG气缸
ORLD
TIMX(550) 0057 D342  ; NG气缸到位延时, NG拨料气缸伸出位延时
; rung 83
LDNOT H3.12  ; 扫码NG气缸原位屏蔽
AND 2.11  ; 扫码NG缸原位
LD H3.12  ; 扫码NG气缸原位屏蔽
AND 7.13  ; 扫码NG缸
ORLD
TIMX(550) 0100 D144  ; 扫码NG缸原位时间, 扫码NG缸延时原位
; rung 84
LDNOT H3.13  ; 扫码NG气缸到位屏蔽
AND 2.12  ; 扫码NG缸到位
LD H3.13  ; 扫码NG气缸到位屏蔽
ANDNOT 7.13  ; 扫码NG缸
ORLD
TIMX(550) 0101 D145  ; 扫码NG缸原位时间, 扫码NG缸延时到位
; rung 85: 1#腔体有料
LD H4.00  ; 1#腔体有料
ORNOT 3.01  ; 腔体1有料
MOV(021) D148 D348  ; 1#腔体有料延时
TIMX(550) 0020 &5  ; 腔体1有料延时

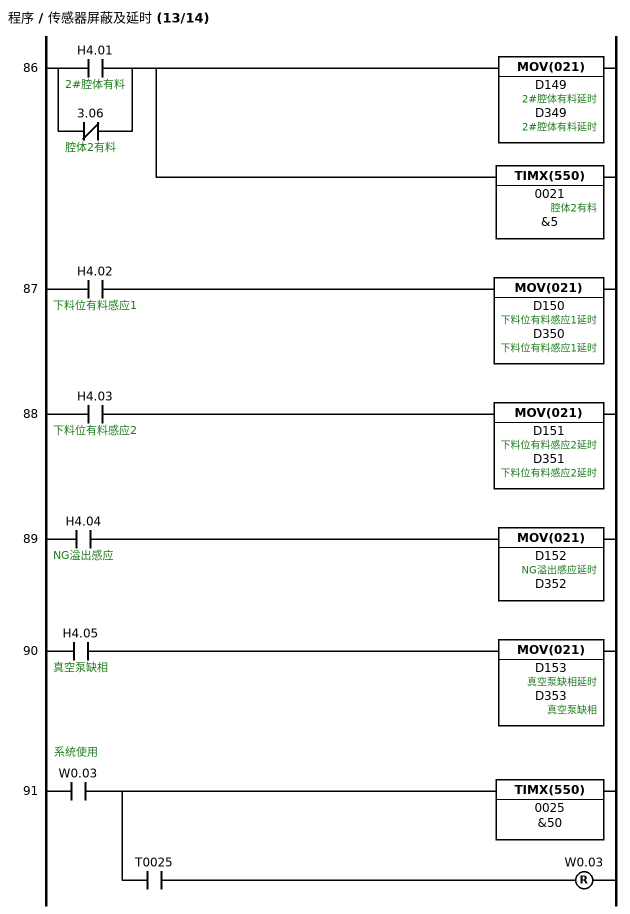
; rung 86
LD H4.01  ; 2#腔体有料
ORNOT 3.06  ; 腔体2有料
MOV(021) D149 D349  ; 2#腔体有料延时
TIMX(550) 0021 &5  ; 腔体2有料
; rung 87
LD H4.02  ; 下料位有料感应1
MOV(021) D150 D350  ; 下料位有料感应1延时
; rung 88
LD H4.03  ; 下料位有料感应2
MOV(021) D151 D351  ; 下料位有料感应2延时
; rung 89
LD H4.04  ; NG溢出感应
MOV(021) D152 D352  ; NG溢出感应延时
; rung 90
LD H4.05  ; 真空泵缺相
MOV(021) D153 D353  ; 真空泵缺相延时, 真空泵缺相
; rung 91: 系统使用
LD W0.03
TIMX(550) 0025 &50
AND T0025
RSET W0.03

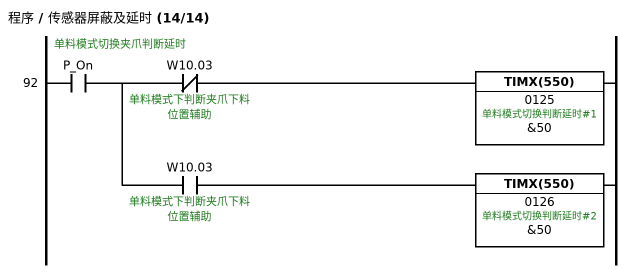
; rung 92: 单料模式切换夹爪判断延时
LD P_On
OUT TR0
ANDNOT W10.03  ; 单料模式下判断夹爪下料位置辅助
TIMX(550) 0125 &50  ; 单料模式切换判断延时#1
LD TR0
AND W10.03  ; 单料模式下判断夹爪下料位置辅助
TIMX(550) 0126 &50  ; 单料模式切换判断延时#2

### Section END
; rung 0
END(001)